# EPICS substitutions: modules/event/evrIoc/Db/bsaSimXL09.substitutions
# Simulation files :
file bsaBPMSTest.db {
  pattern { DEVICE       , S           }
	  { BPMS:XX09:1  , ".1 second" }
	  { BPMS:XX09:2  , ".1 second" }
	  { BPMS:XX09:3  , ".1 second" }
	  { BPMS:XX09:4  , ".1 second" }
	  { BPMS:XX09:5  , ".1 second" }
	  { BPMS:XX09:6  , ".1 second" }
}
file bsaTOROTest.db {
  pattern { DEVICE       , S           }
	  { TORO:XX09:1  , ".1 second" }
	  { TORO:XX09:2  , ".1 second" }
}
# ESIM Pattern records (from EVG) to EVR:
#file evrPatternTest.db {
#  pattern { EIOC  ,  DEVICE }
#	  { IOC:XL09:EV01  ,ESIM:XX09:1  }
#}

# EVG EDEF checking simulation for Modifier5/ bsa enable/disable:
#file bsaProcTestAll.db {
#  pattern {  DEVICE    , LOC     }
#	      { ESIM:XX09:1, SYS0    }
#}
